PROGRAM MAIN
VAR
END_VAR

END_PROGRAM

(* stored: Version 1.1.0.1
   POU MAIN: Id {092a1dda-17e1-41cb-bedf-8a8a9e72da13} *)
